TYPE ST_ErrorInfo EXTENDS ST_SectionBase :
STRUCT
	nErrCode	: UDINT;
	nTotalLen	: BYTE;
	ActChars	: BYTE; //max of 50;
	sErrDescription	:	STRING(50);
	nZeroFill	: BYTE;
END_STRUCT
END_TYPE

(* stored: Version 1.1.0.1, ProductVersion 3.1.4024.12
   DUT ST_ErrorInfo: Id {6a3799eb-120c-4e03-a57c-23d2faa545c8} *)
